FUNCTION_BLOCK FB_RollerDoor
VAR_INPUT
	AutoMode : BOOL;
	ManualMode : BOOL;
	ManualDoorOpenRequest : BOOL;
	ManualDoorCloseRequest : BOOL;
	AutoDoorOpenRequest : BOOL;
	AutoDoorCloseRequest : BOOL;
	test:bool;
END_VAR
VAR_OUTPUT
	DoorOpenCommand : BOOL;
	DoorCloseCommand : BOOL;
END_VAR
VAR
	ManualDoorOpenRequestRTRIG : R_TRIG;
	ManualDoorCloseRequestRTRIG : R_TRIG;
	AutoDoorOpenRequestRTRIG : R_TRIG;
	AutoDoorCloseRequestRTRIG : R_TRIG;
END_VAR

IF AutoMode THEN
	
	AutoDoorOpenRequestRTRIG(CLK := AutoDoorOpenRequest);
	AutoDoorCloseRequestRTRIG(CLK := AutoDoorCloseRequest);
	
	IF AutoDoorOpenRequestRTRIG.Q THEN
		DoorOpenCommand := 1;
		DoorCloseCommand := 0;
	ELSIF AutoDoorCloseRequestRTRIG.Q THEN
		DoorCloseCommand := 1;
		DoorOpenCommand := 0;
	END_IF
END_IF

IF ManualMode THEN
	
	ManualDoorOpenRequestRTRIG(CLK := ManualDoorOpenRequest);
	ManualDoorCloseRequestRTRIG(CLK := ManualDoorCloseRequest);
	
	IF ManualDoorOpenRequestRTRIG.Q THEN
		DoorOpenCommand := 1;
		DoorCloseCommand := 0;
	ELSIF ManualDoorCloseRequestRTRIG.Q THEN
		DoorCloseCommand := 1;
		DoorOpenCommand := 0;
	END_IF
END_IF

END_FUNCTION_BLOCK

(* stored: Version 1.1.0.1, ProductVersion 3.1.4024.12
   POU FB_RollerDoor: Id {0c8919ff-7e11-4bc8-ba75-d10e0a4bf504}, SpecialFunc None *)
